FUNCTION_BLOCK Weighbridge
VAR_INPUT
	Definitions : MOD_WeighBridge_istDefinitions;
	Sensor : MOD_Weighbridge_istSensor;
END_VAR
VAR_OUTPUT
	Output : MOD_WeighBridge_qstOutput;
END_VAR
VAR
	State : INT;
END_VAR

IF Sensor.Weight <= Definitions.OperatingWeight THEN
	Output.TruckOnScale := FALSE;
ELSE
	Output.TruckOnScale := TRUE;	
END_IF

IF Sensor.Weight > Definitions.WeightLimit - Definitions.DetractorWeight THEN
	Output.WeightLimitReached := TRUE;
ELSE
	Output.WeightLimitReached := FALSE;
END_IF

IF FALSE THEN //error stop pause ETC
	Output.WeightLimitReached := FALSE;
	Output.TruckOnScale := FALSE;
END_IF

END_FUNCTION_BLOCK

(* stored: Version 1.1.0.1, ProductVersion 3.1.4024.6
   POU Weighbridge: Id {adb499aa-6201-4292-b9d1-d349fb2c2ab6}, SpecialFunc None *)
